FUNCTION_BLOCK SS3_v_direct (* Composite FB wrapping other FBs *)
  (* Standard: 61499-2 *)
  (* Version 1.0, 2025-05-26, DEVIASH *)
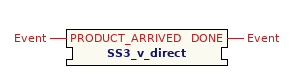
  EVENT_INPUT
    PRODUCT_ARRIVED; (* Initialization Request *)
  END_EVENT
  EVENT_OUTPUT
    DONE; (* Initialization Confirm *)
  END_EVENT
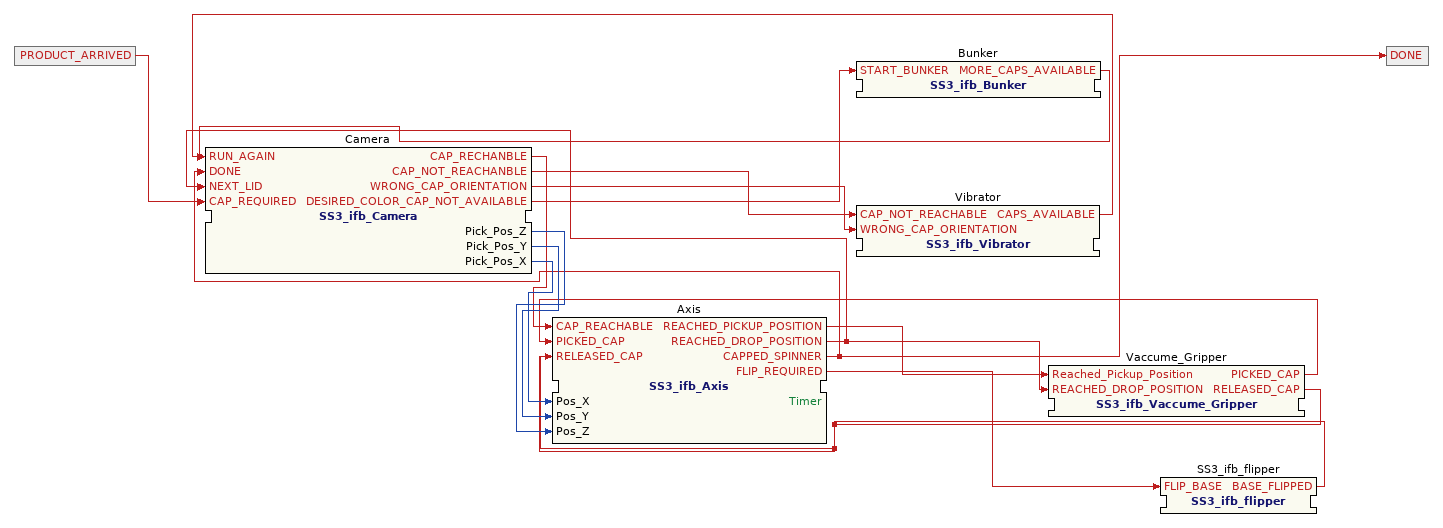
  FBS
    Camera : SS3_ifb_Camera;
    Vaccume_Gripper : SS3_ifb_Vaccume_Gripper;
    Bunker : SS3_ifb_Bunker;
    SS3_ifb_flipper : SS3_ifb_flipper;
    Vibrator : SS3_ifb_Vibrator;
    Axis : SS3_ifb_Axis;
  END_FBS
  EVENT_CONNECTIONS
    Camera.CAP_RECHANBLE TO Axis.CAP_REACHABLE;
    Camera.CAP_NOT_REACHANBLE TO Vibrator.CAP_NOT_REACHABLE;
    Vaccume_Gripper.PICKED_CAP TO Axis.PICKED_CAP;
    Vaccume_Gripper.RELEASED_CAP TO Axis.RELEASED_CAP;
    Camera.WRONG_CAP_ORIENTATION TO Vibrator.WRONG_CAP_ORIENTATION;
    Axis.REACHED_PICKUP_POSITION TO Vaccume_Gripper.Reached_Pickup_Position;
    Vibrator.CAPS_AVAILABLE TO Camera.RUN_AGAIN;
    Axis.REACHED_DROP_POSITION TO Vaccume_Gripper.REACHED_DROP_POSITION;
    Axis.CAPPED_SPINNER TO Camera.DONE;
    Camera.DESIRED_COLOR_CAP_NOT_AVAILABLE TO Bunker.START_BUNKER;
    Bunker.MORE_CAPS_AVAILABLE TO Camera.RUN_AGAIN;
    Axis.REACHED_DROP_POSITION TO Camera.NEXT_LID;
    Axis.FLIP_REQUIRED TO SS3_ifb_flipper.FLIP_BASE;
    SS3_ifb_flipper.BASE_FLIPPED TO Axis.RELEASED_CAP;
    PRODUCT_ARRIVED TO Camera.CAP_REQUIRED;
    Axis.CAPPED_SPINNER TO DONE;
  END_CONNECTIONS
  DATA_CONNECTIONS
    Camera.Pick_Pos_Z TO Axis.Pos_Z;
    Camera.Pick_Pos_Y TO Axis.Pos_Y;
    Camera.Pick_Pos_X TO Axis.Pos_X;
  END_CONNECTIONS
END_FUNCTION_BLOCK
